{attribute 'pack_mode' := '1'}
TYPE ST_ReceiveDataFormat :
STRUCT
   command        : STRING(4);
   seq_number    : ULINT;
   value        : STRING(10240);
END_STRUCT
END_TYPE

(* stored: Version 1.1.0.1, ProductVersion 3.1.4024.15
   DUT ST_ReceiveDataFormat: Id {3c613a2d-c25b-424a-b379-9347d15661a8} *)
